(* IEC 61131-3 sources: com.logicals.lc3.webinar/usRTS_RPMControl_iSOC/src_FB_LIB_SAFE/Numeric/USINT, 8 files *)

(* ---- wADD_USINT_2.iecst ---- *)
NAMESPACE logicals.web.standard
NAMESPACE numeric

/*
 * Function block wrapper for IEC 61131-3 ADD<br>
 * IN1 =  1st value (USINT)<br>
 * IN2 =  2nd value (USINT)<br>
 * OUT = Sum of all input values (USINT)<br>
 */
FUNCTION_BLOCK wADD_USINT_2
	{ vNameAlignment:="center"; altName:="+"; bgColor:="Plum"; width:=40; hideIONames; }
	VAR_INPUT
		IN1 : USINT;
		IN2 : USINT;
	END_VAR
	VAR_OUTPUT
		OUT : USINT;
	END_VAR

	OUT := ADD(IN1:=IN1, IN2:=IN2, ENO=>ENO);
END_FUNCTION_BLOCK

END_NAMESPACE
END_NAMESPACE

(* ---- wADD_USINT_3.iecst ---- *)
NAMESPACE logicals.web.standard
NAMESPACE numeric

/*
 * Function block wrapper for IEC 61131-3 ADD<br>
 * IN1 =  1st value (USINT)<br>
 * IN2 =  2nd value (USINT)<br>
 * IN3 =  3rd value (USINT)<br>
 * OUT = Sum of all input values (USINT)<br>
 */
FUNCTION_BLOCK wADD_USINT_3
	{ vNameAlignment:="center"; altName:="+"; bgColor:="Plum"; width:=40; hideIONames; }
	VAR_INPUT
		IN1 : USINT;
		IN2 : USINT;
		IN3 : USINT;
	END_VAR
	VAR_OUTPUT
		OUT : USINT;
	END_VAR

	OUT := ADD(IN1:=IN1, IN2:=IN2, IN3:=IN3, ENO=>ENO);
END_FUNCTION_BLOCK

END_NAMESPACE
END_NAMESPACE

(* ---- wADD_USINT_4.iecst ---- *)
NAMESPACE logicals.web.standard
NAMESPACE numeric

/*
 * Function block wrapper for IEC 61131-3 ADD<br>
 * IN1 =  1st value (USINT)<br>
 * IN2 =  2nd value (USINT)<br>
 * IN3 =  3rd value (USINT)<br>
 * IN4 =  4th value (USINT)<br>
 * OUT = Sum of all input values (USINT)<br>
 */
FUNCTION_BLOCK wADD_USINT_4
	{ vNameAlignment:="center"; altName:="+"; bgColor:="Plum"; width:=40; hideIONames; }
	VAR_INPUT
		IN1 : USINT;
		IN2 : USINT;
		IN3 : USINT;
		IN4 : USINT;
	END_VAR
	VAR_OUTPUT
		OUT : USINT;
	END_VAR

	OUT := ADD(IN1:=IN1, IN2:=IN2, IN3:=IN3, IN4:=IN4, ENO=>ENO);
END_FUNCTION_BLOCK

END_NAMESPACE
END_NAMESPACE

(* ---- wDIV_USINT.iecst ---- *)
NAMESPACE logicals.web.standard
NAMESPACE numeric

/*
 * Function block wrapper for IEC 61131-3 DIV<br>
 * IN1 =  1st value (USINT)<br>
 * IN2 =  2nd value (USINT)<br>
 * OUT = quotient of IN1 divided by IN2 (USINT)<br>
 */
FUNCTION_BLOCK wDIV_USINT
	{ vNameAlignment:="center"; altName:="/"; bgColor:="Plum"; width:=40; hideIONames; }
	VAR_INPUT
		IN1 : USINT;
		IN2 : USINT;
	END_VAR
	VAR_OUTPUT
		OUT : USINT;
	END_VAR

	OUT := DIV(IN1:=IN1, IN2:=IN2, ENO=>ENO);
END_FUNCTION_BLOCK

END_NAMESPACE
END_NAMESPACE

(* ---- wMUL_USINT_2.iecst ---- *)
NAMESPACE logicals.web.standard
NAMESPACE numeric

/*
 * Function block wrapper for IEC 61131-3 MUL<br>
 * IN1 =  1st value (USINT)<br>
 * IN2 =  2nd value (USINT)<br>
 * OUT = Product of multiplication of all inputs (USINT)<br>
 */
FUNCTION_BLOCK wMUL_USINT_2
	{ vNameAlignment:="center"; altName:="*"; bgColor:="Plum"; width:=40; hideIONames; }
	VAR_INPUT
		IN1 : USINT;
		IN2 : USINT;
	END_VAR
	VAR_OUTPUT
		OUT : USINT;
	END_VAR

	OUT := MUL(IN1:=IN1, IN2:=IN2, ENO=>ENO);
END_FUNCTION_BLOCK

END_NAMESPACE
END_NAMESPACE

(* ---- wMUL_USINT_3.iecst ---- *)
NAMESPACE logicals.web.standard
NAMESPACE numeric

/*
 * Function block wrapper for IEC 61131-3 MUL<br>
 * IN1 =  1st value (USINT)<br>
 * IN2 =  2nd value (USINT)<br>
 * IN3 =  3rd value (USINT)<br>
 * OUT = Product of multiplication of all inputs (USINT)<br>
 */
FUNCTION_BLOCK wMUL_USINT_3
	{ vNameAlignment:="center"; altName:="*"; bgColor:="Plum"; width:=40; hideIONames; }
	VAR_INPUT
		IN1 : USINT;
		IN2 : USINT;
		IN3 : USINT;
	END_VAR
	VAR_OUTPUT
		OUT : USINT;
	END_VAR

	OUT := MUL(IN1:=IN1, IN2:=IN2, IN3:=IN3, ENO=>ENO);
END_FUNCTION_BLOCK

END_NAMESPACE
END_NAMESPACE

(* ---- wMUL_USINT_4.iecst ---- *)
NAMESPACE logicals.web.standard
NAMESPACE numeric

/*
 * Function block wrapper for IEC 61131-3 MUL<br>
 * IN1 =  1st value (USINT)<br>
 * IN2 =  2nd value (USINT)<br>
 * IN3 =  3rd value (USINT)<br>
 * IN4 =  4th value (USINT)<br>
 * OUT = Product of multiplication of all inputs (USINT)<br>
 */
FUNCTION_BLOCK wMUL_USINT_4
	{ vNameAlignment:="center"; altName:="*"; bgColor:="Plum"; width:=40; hideIONames; }
	VAR_INPUT
		IN1 : USINT;
		IN2 : USINT;
		IN3 : USINT;
		IN4 : USINT;
	END_VAR
	VAR_OUTPUT
		OUT : USINT;
	END_VAR

	OUT := MUL(IN1:=IN1, IN2:=IN2, IN3:=IN3, IN4:=IN4, ENO=>ENO);
END_FUNCTION_BLOCK

END_NAMESPACE
END_NAMESPACE

(* ---- wSUB_USINT.iecst ---- *)
NAMESPACE logicals.web.standard
NAMESPACE numeric

/*
 * Function block wrapper for IEC 61131-3 SUB<br>
 * IN1 =  1st value (USINT)<br>
 * IN2 =  2nd value (USINT)<br>
 * OUT = IN1 minus IN2 (USINT)<br>
 */
FUNCTION_BLOCK wSUB_USINT
	{ vNameAlignment:="center"; altName:="-"; bgColor:="Plum"; width:=40; hideIONames; }
	VAR_INPUT
		IN1 : USINT;
		IN2 : USINT;
	END_VAR
	VAR_OUTPUT
		OUT : USINT;
	END_VAR

	OUT := SUB(IN1:=IN1, IN2:=IN2, ENO=>ENO);
END_FUNCTION_BLOCK

END_NAMESPACE
END_NAMESPACE
